PROGRAM MAIN
VAR
	number : int;
END_VAR

END_PROGRAM

(* stored: Version 1.1.0.1, ProductVersion 3.1.4024.12
   POU MAIN: Id {acf28d03-1936-483a-8d10-64cea9f780e8}, SpecialFunc None *)
